FUNCTION "FC_SimReceivingPit" : Void
{ S7_Optimized_Access := 'TRUE' }
VERSION : 1.0
// ==============================================================================
// FC_SimReceivingPit - Ð¡Ð¸Ð¼ÑƒÐ»ÑÑ‚Ð¾Ñ€ Ð¿Ñ€Ð¸Ð¹Ð¼Ð°Ð»ÑŒÐ½Ð¾Ñ— ÑÐ¼Ð¸ (Ð·Ð°Ð³Ð»ÑƒÑˆÐºÐ°)
// ==============================================================================
// Ð’ÐµÑ€ÑÑ–Ñ: 1.0.0
// Ð”Ð°Ñ‚Ð°: 2026-03-24
// ==============================================================================
// ÐŸÑ€Ð¸Ð·Ð½Ð°Ñ‡ÐµÐ½Ð½Ñ:
//   Ð—Ð°Ð³Ð»ÑƒÑˆÐºÐ° Ð´Ð»Ñ ÑƒÐ½Ð¸ÐºÐ½ÐµÐ½Ð½Ñ Ð¿Ð¾Ð¼Ð¸Ð»Ð¾Ðº Ð¿Ñ€Ð¸ ÐºÐ¾Ð¼Ð¿Ñ–Ð»ÑÑ†Ñ–Ñ—
//   Ð ÐµÐ°Ð»ÑŒÐ½Ð° Ñ„ÑƒÐ½ÐºÑ†Ñ–Ð¾Ð½Ð°Ð»ÑŒÐ½Ñ–ÑÑ‚ÑŒ Ð¼Ð¾Ð¶Ðµ Ð±ÑƒÑ‚Ð¸ Ð´Ð¾Ð´Ð°Ð½Ð° Ð¿Ñ–Ð·Ð½Ñ–ÑˆÐµ
// ==============================================================================
   VAR_INPUT
      ReceivingPitIdx : Int;   // Ñ–Ð½Ð´ÐµÐºÑ Ñƒ DB_Mechs.ReceivingPit[]
      Enable : Bool;   // ÑƒÐ²Ñ–Ð¼ÐºÐ½ÑƒÑ‚Ð¸ ÑÐ¸Ð¼ÑƒÐ»ÑÑ†Ñ–ÑŽ
   END_VAR


BEGIN

	// === Ð—ÐÐ“Ð£Ð›Ð¨ÐšÐ ===
	// Ð ÐµÐ°Ð»ÑŒÐ½Ð° Ñ„ÑƒÐ½ÐºÑ†Ñ–Ð¾Ð½Ð°Ð»ÑŒÐ½Ñ–ÑÑ‚ÑŒ Ð±ÑƒÐ´Ðµ Ð´Ð¾Ð´Ð°Ð½Ð° Ð¿Ñ–Ð·Ð½Ñ–ÑˆÐµ
	// ÐÐ°Ñ€Ð°Ð·Ñ– Ð¿Ñ€Ð¾ÑÑ‚Ð¾ ÑƒÐ½Ð¸ÐºÐ°Ñ”Ð¼Ð¾ Ð¿Ð¾Ð¼Ð¸Ð»Ð¾Ðº Ð¿Ñ€Ð¸ Ð²Ð¸ÐºÐ»Ð¸ÐºÑƒ

	// ÐŸÐµÑ€ÐµÐ²Ñ–Ñ€ÐºÐ° Ñ–Ð½Ð´ÐµÐºÑÑƒ (Ñ‰Ð¾Ð± ÑƒÐ½Ð¸ÐºÐ½ÑƒÑ‚Ð¸ OOB)
	IF #ReceivingPitIdx > "RECEIVING_PITS_COUNT" THEN
	    RETURN;
	END_IF;

	// Ð¢ÑƒÑ‚ Ð±ÑƒÐ´Ðµ Ð»Ð¾Ð³Ñ–ÐºÐ° ÑÐ¸Ð¼ÑƒÐ»ÑÑ†Ñ–Ñ— Ð¿Ñ€Ð¸Ð¹Ð¼Ð°Ð»ÑŒÐ½Ð¾Ñ— ÑÐ¼Ð¸:
	// - Ð¡Ð¸Ð¼ÑƒÐ»ÑÑ†Ñ–Ñ Ð·Ð²Ð¾Ñ€Ð¾Ñ‚Ð½Ð¾Ð³Ð¾ Ð·Ð²'ÑÐ·ÐºÑƒ
	// - Ð¡Ð¸Ð¼ÑƒÐ»ÑÑ†Ñ–Ñ Ð°Ð²Ð°Ñ€Ñ–Ð¹


END_FUNCTION

